PROGRAM main
VAR
	bt_start_t1 AT %IX0.0 : bool;
	bt_stop_t1 AT %IX0.1 : bool;
	bt_emerg_t1 AT %IX0.2 : bool;
	led_start_t1 AT %QX0.0 : bool;
	led_stop_t1 AT %QX0.1 : bool;
	nivel_t1 AT %IW0 : int;
	vazao_t1 AT %IW1 : int;
	valv_entrada_t1 AT %QW0 : int;
	valv_saida_t1 AT %QW1 : int;
	display_t1 AT %QW2 : int;
	bt_start_t2 AT %IX0.4 : bool;
	bt_stop_t2 AT %IX0.5 : bool;
	bt_emerg_t2 AT %IX0.6 : bool;
	led_start_t2 AT %QX0.2 : bool;
	nivel_t2 AT %IW4 : int;
	valv_entrada_t2 AT %QW4 : int;
	valv_saida_t2 AT %QW5 : int;
	display_t2 AT %QW6 : int;
	mem_start_t1 : bool;
	mem_start_t2 : bool;
	cmd_fill_t1 AT %QX2.0 : bool;
	cmd_drain_t1 AT %QX2.1 : bool := 0;
	cmd_fill_t2 AT %QX2.2 : bool;
	cmd_drain_t2 AT %QX2.3 : bool := 0;
	cmd_remote AT %QX2.4 : bool;
	flag_val_t1 : bool;
	flag_val_t2 : bool;
	flag_drain_t1 : bool;
	flag_drain_t2 : bool;
END_VAR

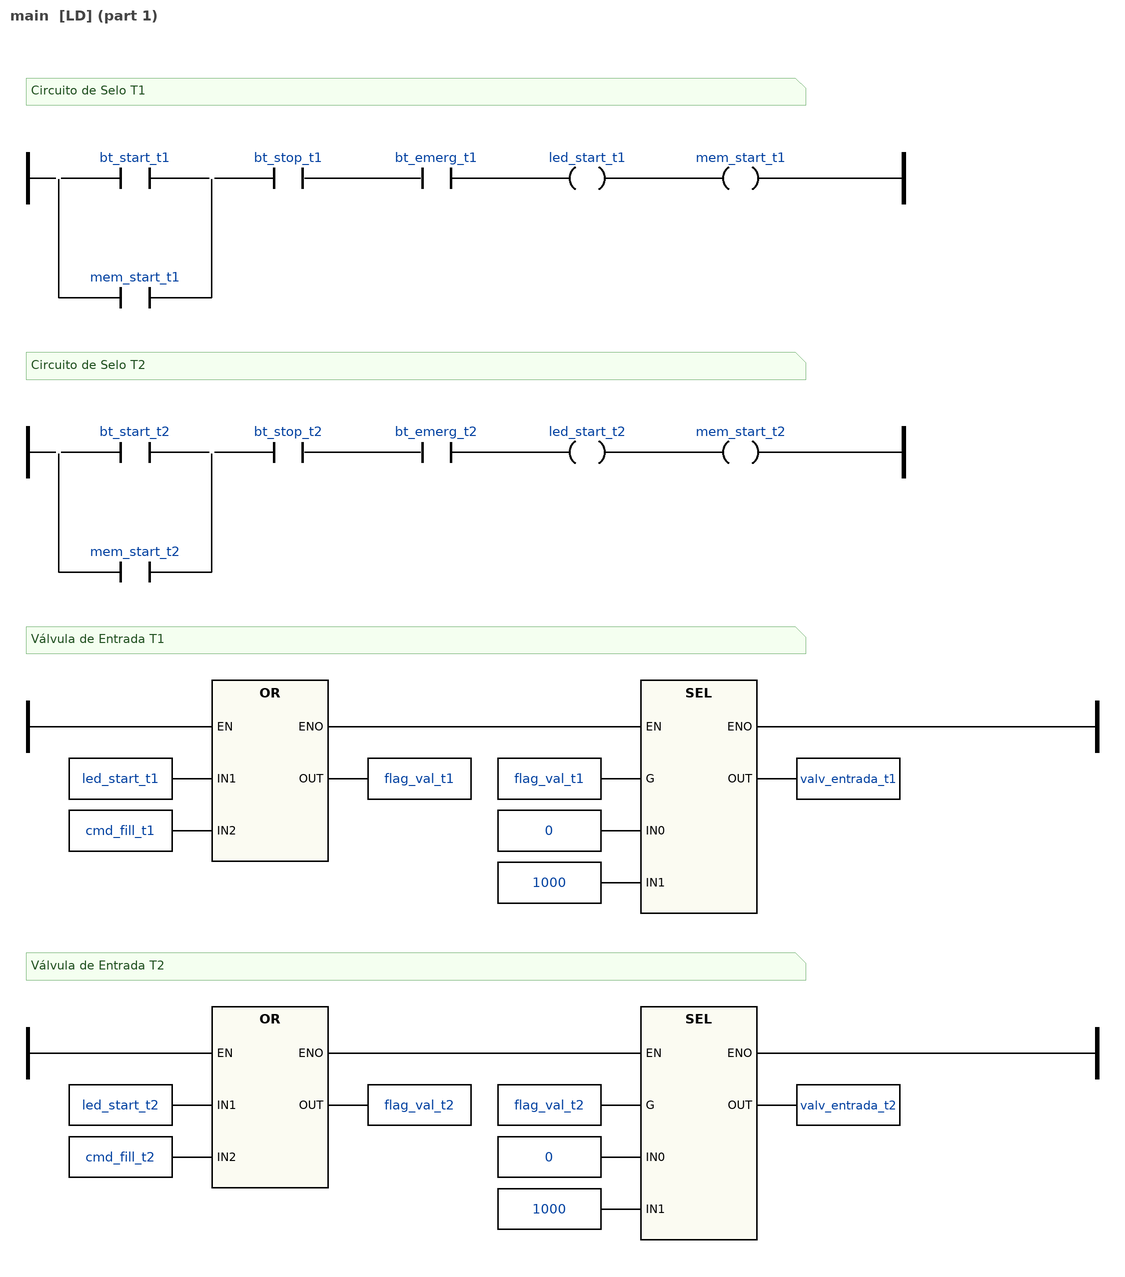
(* LD diagram, written out as Structured Text *)
(* Circuito de Selo T1 *)
led_start_t1 := (bt_start_t1 OR mem_start_t1) AND bt_stop_t1 AND bt_emerg_t1;
mem_start_t1 := (bt_start_t1 OR mem_start_t1) AND bt_stop_t1 AND bt_emerg_t1;
(* Circuito de Selo T2 *)
led_start_t2 := (bt_start_t2 OR mem_start_t2) AND bt_stop_t2 AND bt_emerg_t2;
mem_start_t2 := (bt_start_t2 OR mem_start_t2) AND bt_stop_t2 AND bt_emerg_t2;
(* Válvula de Entrada T1 *)
flag_val_t1 := led_start_t1 OR cmd_fill_t1;
valv_entrada_t1 := SEL(flag_val_t1, 0, 1000);
(* Válvula de Entrada T2 *)
flag_val_t2 := led_start_t2 OR cmd_fill_t2;
valv_entrada_t2 := SEL(flag_val_t2, 0, 1000);
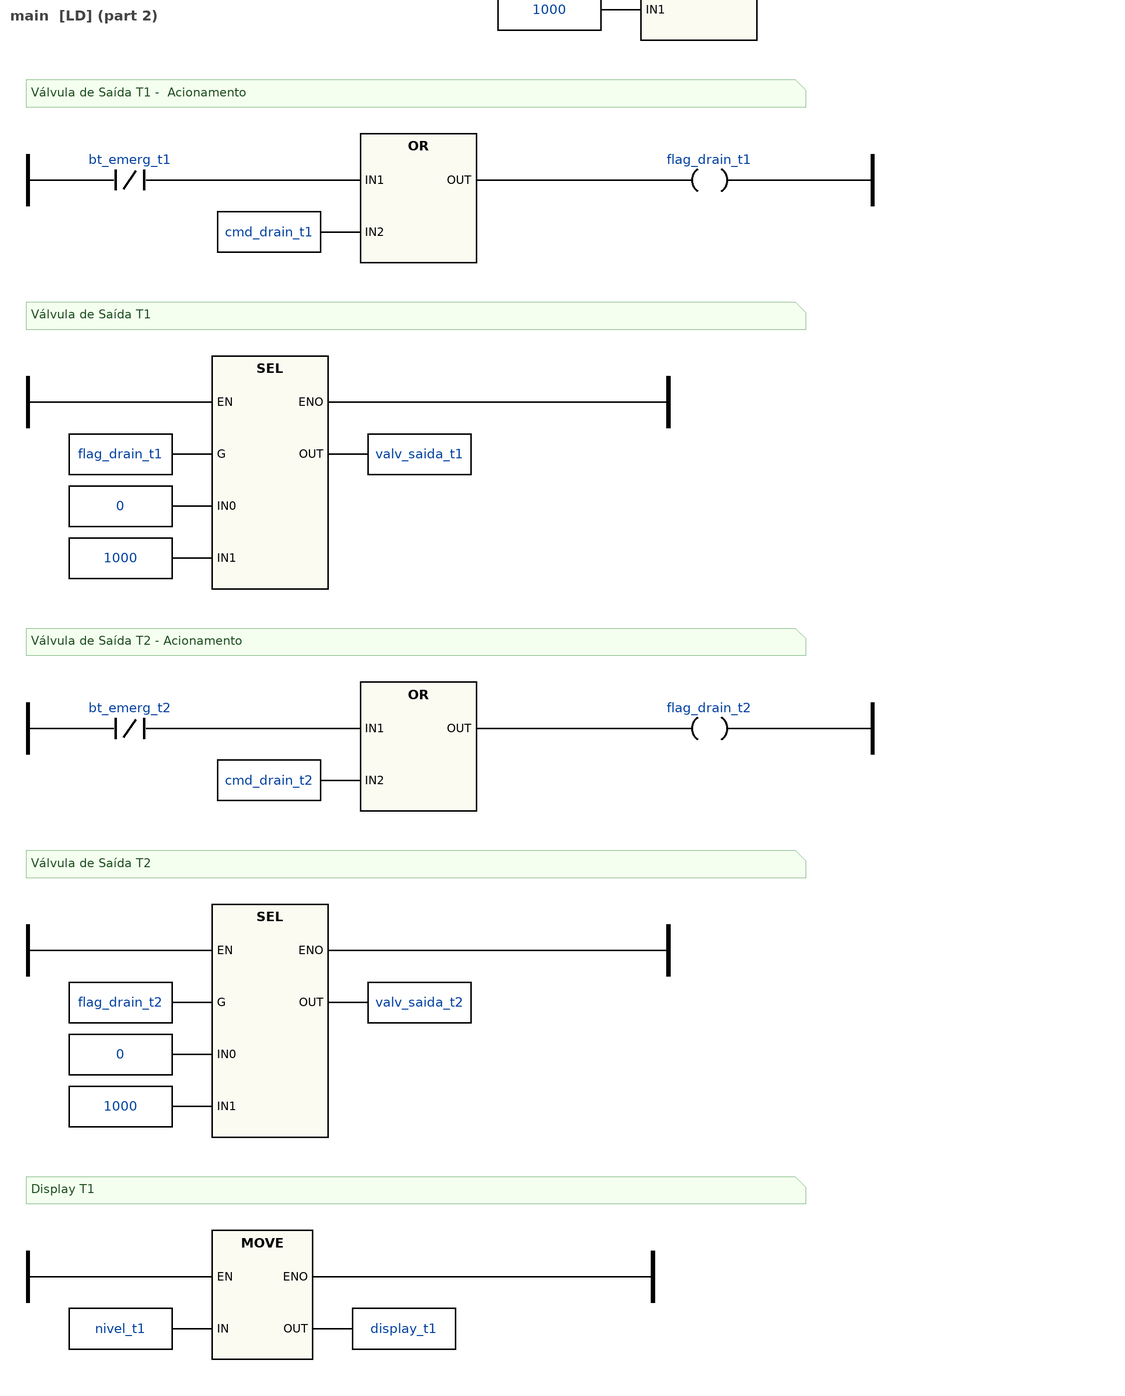
(* Válvula de Saída T1 -  Acionamento *)
flag_drain_t1 := NOT bt_emerg_t1 OR cmd_drain_t1;
(* Válvula de Saída T1 *)
valv_saida_t1 := SEL(flag_drain_t1, 0, 1000);
(* Válvula de Saída T2 - Acionamento *)
flag_drain_t2 := NOT bt_emerg_t2 OR cmd_drain_t2;
(* Válvula de Saída T2 *)
valv_saida_t2 := SEL(flag_drain_t2, 0, 1000);
(* Display T1 *)
display_t1 := nivel_t1;
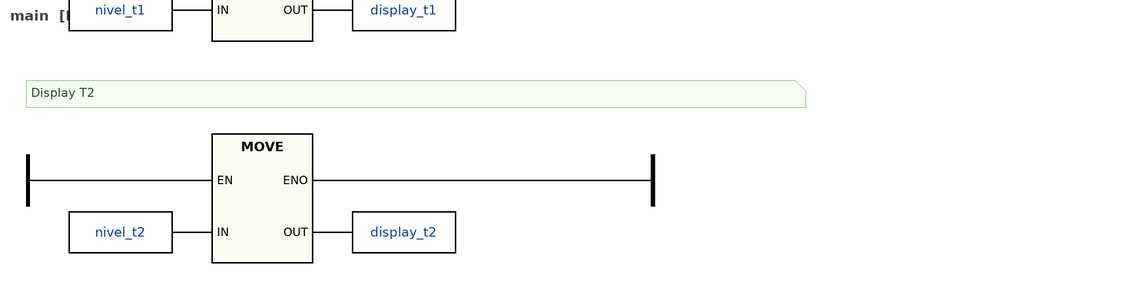
(* Display T2 *)
display_t2 := nivel_t2;
END_PROGRAM
